(* IEC 61131-3 sources: CodesysTest/export/ObjectHandling/FB_CollectionHandlerPositionableMotors.pou, 2 files *)

(* ---- FB_CollectionHandlerPositionableMotors.pou.st ---- *)
(*#-#-#-#-#-#-#-#-#-#---Declaration---#-#-#-#-#-#-#-#-#-#-#-#-#*)

FUNCTION_BLOCK FB_CollectionHandlerPositionableMotors
VAR_INPUT
END_VAR
VAR
	Collection: ARRAY[0..GlobalObjects.MAX_MOTORS] OF IPositionableMotor; // object array
	ObjNames   : ARRAY[0..GlobalObjects.MAX_MOTORS] OF STRING;
	_ArrayOver   : BOOL;
	_BadObj      : INT;
	_DupeObj   : INT;
	_OverObj   : INT;
	_TotalObj   : UINT;
END_VAR(*#-#-#-#-#-#-#-#-#-#---Implementation---#-#-#-#-#-#-#-#-#-#-#-#-#*)

(* ---- AddObject.m.st ---- *)
(*#-#-#-#-#-#-#-#-#-#---Declaration---#-#-#-#-#-#-#-#-#-#-#-#-#*)

METHOD AddObject
VAR_INPUT
	Obj   : IPositionableMotor;
END_VAR
VAR
	J   : UINT;
END_VAR(*#-#-#-#-#-#-#-#-#-#---Implementation---#-#-#-#-#-#-#-#-#-#-#-#-#*)

FOR J:= 0 TO _TotalObj DO
	IF Collection[J] = Obj THEN
		// object pointer matches - dupe!
		_DupeObj:= _DupeObj + 1;
		RETURN;
	END_IF
END_FOR

IF _TotalObj < GlobalObjects.MAX_MOTORS THEN
	Collection[_TotalObj]:= Obj;
	ObjNames[_TotalObj]:= Obj.InstanceName;
	_TotalObj:= _TotalObj + 1;
ELSE
	_ArrayOver:= TRUE;
	_OverObj:= _OverObj + 1;
END_IF
